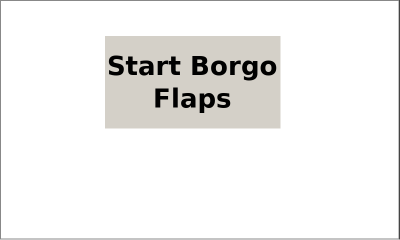
VISUALIZATION V_ProductionBorgoFlaps  // 400x240
VAR_IN_OUT
	HMI : ST_PackMLBaseModule_HMI;
END_VAR
    RoundedRectangle (0,-1 400x240)
    RoundedRectangle (105,36 175x92), "Start Borgo Flaps"
        OnMouseClick: execute { HMI.Command.State := E_PMLCommand.ePMLCommand_Start; }
END_VISUALIZATION

(* stored: Version 1.1.0.1, ProductVersion 3.1.4024.15
   Visu V_ProductionBorgoFlaps: Id {571e1921-2ea2-4d68-a038-db63e03e77f7} *)
